TYPE ST_OvercurrentProtection_set :
STRUCT
	ui_PowerlockInputCurrentLimit			: ARRAY [1..2] OF UINT := [400,400];
	ui_PowerlockOutputCurrentLimit			: ARRAY [1..3] OF UINT := [400,400,400];
END_STRUCT
END_TYPE

(* stored: Version 1.1.0.1, ProductVersion 3.1.4026.18
   DUT ST_OvercurrentProtection_set: Id {01ca00b9-7de0-4b90-be2a-3f4bd792f1db} *)
